TEXTLIST M2AxesTextList
  0 = 'X (010)'
  1 = 'Y (100)'
  2 = 'Z (000)'
  3 = 'Tilt X (001)'
  4 = 'Tilt Y (110)'
   = ''
END_TEXTLIST

(* stored: Version 1.1.0.1, ProductVersion 3.1.4018.5
   TextList M2AxesTextList: Id {c9947a1d-e7d6-4adb-83aa-155db8e3bce2} *)
